(* PLC project Practical Work One, Rexroth ctrlX PLC Engineering ctrlX PLC 1.16.1, author Cedric Lenoir *)
(* stored: creationDateTime 2024-02-07T14:58:28.9317925, version 0.0, modificationDateTime 2024-02-07T14:56:44.3352338, organization HEVS *)
(* First Test for Practical Work One *)

TYPE UA_DigitalInput_32 : STRUCT
  Input_0_0 : BOOL;
  Input_0_1 : BOOL;
  Input_0_2 : BOOL;
  Input_0_3 : BOOL;
  Input_0_4 : BOOL;
  Input_0_5 : BOOL;
  Input_0_6 : BOOL;
  Input_0_7 : BOOL;
  Input_1_0 : BOOL;
  Input_1_1 : BOOL;
  Input_1_2 : BOOL;
  Input_1_3 : BOOL;
  Input_1_4 : BOOL;
  Input_1_5 : BOOL;
  Input_1_6 : BOOL;
  Input_1_7 : BOOL;
  Input_2_0 : BOOL;
  Input_2_1 : BOOL;
  Input_2_2 : BOOL;
  Input_2_3 : BOOL;
  Input_2_4 : BOOL;
  Input_2_5 : BOOL;
  Input_2_6 : BOOL;
  Input_2_7 : BOOL;
  Input_3_0 : BOOL;
  Input_3_1 : BOOL;
  Input_3_2 : BOOL;
  Input_3_3 : BOOL;
  Input_3_4 : BOOL;
  Input_3_5 : BOOL;
  Input_3_6 : BOOL;
  Input_3_7 : BOOL;
END_STRUCT;
END_TYPE

TYPE UA_DigitalOutput_32 : STRUCT
  Output_0_0 : BOOL;
  Output_0_1 : BOOL;
  Output_0_2 : BOOL;
  Output_0_3 : BOOL;
  Output_0_4 : BOOL;
  Output_0_5 : BOOL;
  Output_0_6 : BOOL;
  Output_0_7 : BOOL;
  Output_1_0 : BOOL;
  Output_1_1 : BOOL;
  Output_1_2 : BOOL;
  Output_1_3 : BOOL;
  Output_1_4 : BOOL;
  Output_1_5 : BOOL;
  Output_1_6 : BOOL;
  Output_1_7 : BOOL;
  Output_2_0 : BOOL;
  Output_2_1 : BOOL;
  Output_2_2 : BOOL;
  Output_2_3 : BOOL;
  Output_2_4 : BOOL;
  Output_2_5 : BOOL;
  Output_2_6 : BOOL;
  Output_2_7 : BOOL;
  Output_3_0 : BOOL;
  Output_3_1 : BOOL;
  Output_3_2 : BOOL;
  Output_3_3 : BOOL;
  Output_3_4 : BOOL;
  Output_3_5 : BOOL;
  Output_3_6 : BOOL;
  Output_3_7 : BOOL;
END_STRUCT;
END_TYPE

TYPE UA_ButtonAndSignal : STRUCT
  In_Estop : BOOL;
  In_Reset : BOOL;
  In_Start : BOOL;
  In_Stop : BOOL;
  Out_Idle : BOOL;
  Out_Execute : BOOL;
  Out_Stopped : BOOL;
END_STRUCT;
END_TYPE

TYPE UA_O300_DL : STRUCT
  Value : WORD;
  BCD1 : BOOL;
  Q : BOOL;
  A : BOOL;
END_STRUCT;
END_TYPE

TYPE UA_O300_ZL : STRUCT
  BCD1 : BOOL;
  Q : BOOL;
  A : BOOL;
END_STRUCT;
END_TYPE

TYPE UA_U300_D50 : STRUCT
  Value : DWORD;
  Scale : SINT;
  SSC1 : BOOL;
  SSC2 : BOOL;
  Q : BOOL;
  A : BOOL;
  SSC4 : BOOL;
END_STRUCT;
END_TYPE

(* www.hevs.ch Institut Systemes Industriels Project: Projet No: PW_01 Author: Cedric Lenoir Date: 2023 October 11 Summary: List of of components for a station of a conveyor. *)
TYPE ST_StationConveyor : STRUCT
  bButton : BOOL;
  bLed : BOOL;
  bSensor : BOOL;
END_STRUCT;
END_TYPE

(* www.hevs.ch Institut Systemes Industriels Project: Projet No: PW_01 Author: Cedric Lenoir Date: 2023 October 11 Summary: List of of components for a motor of a conveyor. *)
TYPE ST_BuzzerConveyor : STRUCT
  bActivate : BOOL;
  tTime : TIME := TIME#2s0ms;
END_STRUCT;
END_TYPE

(* www.hevs.ch Institut Systemes Industriels Project: Projet No: PW_01 Author: Cedric Lenoir Date: 2023 October 11 Summary: List of of components for a motor of a conveyor. *)
TYPE ST_MotorConveyor : STRUCT
  bK_ActivatePositiveDirection : BOOL;
  bK_ActivateNegativeDirection : BOOL;
END_STRUCT;
END_TYPE

TYPE ST_Conveyor : STRUCT
  StationOne : ST_StationConveyor;
  StationTwo : ST_StationConveyor;
  StationThree : ST_StationConveyor;
  StationOutput : ST_StationConveyor;
  Motor : ST_MotorConveyor;
  Buzzer : ST_BuzzerConveyor;
END_STRUCT;
END_TYPE

TYPE ST_HmiConveyor : STRUCT
  bStartConveyor : BOOL;
  bStopConveyor : BOOL;
END_STRUCT;
END_TYPE

TYPE UA_U300_P50 : STRUCT
  Value : DWORD;
  Scale : SINT;
  SSC1 : BOOL;
  SSC2 : BOOL;
  Q : BOOL;
  A : BOOL;
  SSC4 : BOOL;
END_STRUCT;
END_TYPE

TYPE UA_Schunk_mms : STRUCT
  Value : WORD;
END_STRUCT;
END_TYPE

TYPE UA_Balluf_bcm0002 : STRUCT
  Data_1 : REAL;
  Data_2 : REAL;
  Data_3 : REAL;
  Temperature : REAL;
  Status : DWORD;
END_STRUCT;
END_TYPE

TYPE UA_Festo : STRUCT
  SetOut : BOOL;
END_STRUCT;
END_TYPE

TYPE UA_AnalogIn : STRUCT
  IW_04 : WORD;
  IW_06 : WORD;
  IW_08 : WORD;
  IW_10 : WORD;
  IW_12 : WORD;
  IW_14 : WORD;
  IW_16 : WORD;
  IW_18 : WORD;
END_STRUCT;
END_TYPE

TYPE UA_AnalogOut : STRUCT
  QW_04 : WORD;
  QW_06 : WORD;
  QW_08 : WORD;
  QW_10 : WORD;
END_STRUCT;
END_TYPE

TYPE UA_AboxInterface : STRUCT
  uaButtonAndSignal : UA_ButtonAndSignal;
  uaAnalogIn : UA_AnalogIn;
  uaAnalogOut : UA_AnalogOut;
  uaDigitalIn : UA_DigitalInput_32;
  uaDigitalOut : UA_DigitalOutput_32;
  uaO300_DL_Optic : UA_O300_DL;
  uaO300_ZL_Optic : UA_O300_ZL;
  uaU300_D50_Sound : UA_U300_D50;
  uaU300_P50_Sound : UA_U300_P50;
  uaSchunk : UA_Schunk_mms;
  uaSchunkGripper : UA_Festo;
  uaAccelerometer : UA_Balluf_bcm0002;
END_STRUCT;
END_TYPE

TYPE ST_ConveyorTagsIn : STRUCT
  S1_Pb_Station_1 : BOOL;  (* %I0.0 *)
  S2_Pb_Station_2 : BOOL;  (* %I0.1 *)
  S3_Pb_Station_3 : BOOL;  (* %I0.2 *)
  S4_Pb_OutputConveyor : BOOL;  (* %I0.3 *)
  B1_SensorActive : BOOL;  (* %I0.4 *)
  B2_SensorActive : BOOL;  (* %I0.5 *)
  B3_SensorActive : BOOL;  (* %I0.6 *)
  B4_OutputConveyorFree : BOOL;  (* %I0.7 *)
END_STRUCT;
END_TYPE

TYPE ST_ConveyorTagsOut : STRUCT
  H1_LedStation_1 : BOOL;  (* %Q0.0 *)
  H2_LedStation_2 : BOOL;  (* %Q0.1 *)
  H3_LedStation_3 : BOOL;  (* %Q0.2 *)
  H4_LedOutputConveyor : BOOL;  (* %Q0.3 *)
  K1_DirectionOutput : BOOL;  (* %Q0.4 *)
  K2_DirectionH1 : BOOL;  (* %Q0.5 *)
  Buzzer : BOOL;  (* %Q0.6 *)
END_STRUCT;
END_TYPE

(* www.hevs.ch Institut Systemes Industriels Project: Projet No: PW_01 Author: Cedric Lenoir Date: 2023 October 11 Summary: PLC Hello World ! *)
PROGRAM PLC_PRG
  VAR
    iCount : INT := 3;
    TagIn : ST_ConveyorTagsIn;
    TagOut : ST_ConveyorTagsOut;
    rTrigStart : R_TRIG;
    rTrigStop : R_TRIG;
    tonBuzzer : TON;
  END_VAR

                    iCount := iCount + 1;

GetInput();

(*
	Declaration of all FB at the end of the code, this is a good practice.
	You can lose one cycle but the program is more readable.

    But !
    Triggers are exceptions:
        because the output .Q is only active in the current cycle
*)
rTrigStart(CLK:=GVL_Abox.uaAboxInterface.uaButtonAndSignal.In_Start);
rTrigStop(CLK:=GVL_Abox.uaAboxInterface.uaButtonAndSignal.In_Stop);

IF rTrigStart.Q THEN
	TagOut.K1_DirectionOutput := TRUE;
END_IF

IF rTrigStop.Q THEN
	TagOut.K1_DirectionOutput := FALSE;
END_IF

// If Start activated for more than 3 seconds, then Buzzer
tonBuzzer(IN := GVL_Abox.uaAboxInterface.uaButtonAndSignal.In_Start,
	      PT := T#3S);
		  
TagOut.Buzzer := tonBuzzer.Q;

SetOutput();
                  

METHOD GetInput
                          TagIn.S1_Pb_Station_1 := GVL_Abox.uaAboxInterface.uaDigitalIn.Input_0_0;
TagIn.S2_Pb_Station_2 := GVL_Abox.uaAboxInterface.uaDigitalIn.Input_0_1;
TagIn.S3_Pb_Station_3 := GVL_Abox.uaAboxInterface.uaDigitalIn.Input_0_2;
TagIn.S4_Pb_OutputConveyor := GVL_Abox.uaAboxInterface.uaDigitalIn.Input_0_3;

TagIn.B1_SensorActive := GVL_Abox.uaAboxInterface.uaDigitalIn.Input_0_4;
TagIn.B2_SensorActive := GVL_Abox.uaAboxInterface.uaDigitalIn.Input_0_5;
TagIn.B3_SensorActive := GVL_Abox.uaAboxInterface.uaDigitalIn.Input_0_6;
TagIn.B4_OutputConveyorFree := GVL_Abox.uaAboxInterface.uaDigitalIn.Input_0_7;
                        
END_METHOD

METHOD SetOutput
                          GVL_Abox.uaAboxInterface.uaDigitalOut.Output_0_0 := TagOut.H1_LedStation_1;
GVL_Abox.uaAboxInterface.uaDigitalOut.Output_0_1 := TagOut.H2_LedStation_2;
GVL_Abox.uaAboxInterface.uaDigitalOut.Output_0_2 := TagOut.H3_LedStation_3;
GVL_Abox.uaAboxInterface.uaDigitalOut.Output_0_3 := TagOut.H4_LedOutputConveyor;
GVL_Abox.uaAboxInterface.uaDigitalOut.Output_0_4 := TagOut.K1_DirectionOutput;
GVL_Abox.uaAboxInterface.uaDigitalOut.Output_0_5 := TagOut.K2_DirectionH1;
GVL_Abox.uaAboxInterface.uaDigitalOut.Output_0_6 := TagOut.Buzzer;
                        
END_METHOD
END_PROGRAM

PROGRAM PRG_MapBox
  VAR
    UA_ReadCounterFromStation : DINT;  (* Write from Siemens to ctrX Core Used to check if read is running *)
    UA_ButtonAndSignal_In_Estop : BOOL;
    UA_ButtonAndSignal_In_Reset : BOOL;
    UA_ButtonAndSignal_In_Start : BOOL;
    UA_ButtonAndSignal_In_Stop : BOOL;
    UA_Balluf_bcm0002_Data_1 : REAL;
    UA_Balluf_bcm0002_Data_2 : REAL;
    UA_Balluf_bcm0002_Data_3 : REAL;
    UA_Balluf_bcm0002_Temperature : REAL;
    UA_Balluf_bcm0002_Status : DWORD;
    UA_Festo_SetOut : BOOL;
    UA_O300_DL_Value : WORD;
    UA_O300_DL_BCD1 : BOOL;
    UA_O300_DL_Q : BOOL;
    UA_O300_DL_A : BOOL;
    UA_O300_ZL_BCD1 : BOOL;
    UA_O300_ZL_Q : BOOL;
    UA_O300_ZL_A : BOOL;
    UA_U300_D50_Value : DWORD;
    UA_U300_D50_Scale : SINT;
    UA_U300_D50_SSC1 : BOOL;
    UA_U300_D50_SSC2 : BOOL;
    UA_U300_D50_Q : BOOL;
    UA_U300_D50_A : BOOL;
    UA_U300_D50_SSC4 : BOOL;
    UA_U300_P50_Value : DWORD;
    UA_U300_P50_Scale : SINT;
    UA_U300_P50_SSC1 : BOOL;
    UA_U300_P50_SSC2 : BOOL;
    UA_U300_P50_Q : BOOL;
    UA_U300_P50_A : BOOL;
    UA_U300_P50_SSC4 : BOOL;
    UA_DigitalInput_32_Input_0_0 : BOOL;
    UA_DigitalInput_32_Input_0_1 : BOOL;
    UA_DigitalInput_32_Input_0_2 : BOOL;
    UA_DigitalInput_32_Input_0_3 : BOOL;
    UA_DigitalInput_32_Input_0_4 : BOOL;
    UA_DigitalInput_32_Input_0_5 : BOOL;
    UA_DigitalInput_32_Input_0_6 : BOOL;
    UA_DigitalInput_32_Input_0_7 : BOOL;
    UA_DigitalInput_32_Input_1_0 : BOOL;
    UA_DigitalInput_32_Input_1_1 : BOOL;
    UA_DigitalInput_32_Input_1_2 : BOOL;
    UA_DigitalInput_32_Input_1_3 : BOOL;
    UA_DigitalInput_32_Input_1_4 : BOOL;
    UA_DigitalInput_32_Input_1_5 : BOOL;
    UA_DigitalInput_32_Input_1_6 : BOOL;
    UA_DigitalInput_32_Input_1_7 : BOOL;
    UA_DigitalInput_32_Input_2_0 : BOOL;
    UA_DigitalInput_32_Input_2_1 : BOOL;
    UA_DigitalInput_32_Input_2_2 : BOOL;
    UA_DigitalInput_32_Input_2_3 : BOOL;
    UA_DigitalInput_32_Input_2_4 : BOOL;
    UA_DigitalInput_32_Input_2_5 : BOOL;
    UA_DigitalInput_32_Input_2_6 : BOOL;
    UA_DigitalInput_32_Input_2_7 : BOOL;
    UA_DigitalInput_32_Input_3_0 : BOOL;
    UA_DigitalInput_32_Input_3_1 : BOOL;
    UA_DigitalInput_32_Input_3_2 : BOOL;
    UA_DigitalInput_32_Input_3_3 : BOOL;
    UA_DigitalInput_32_Input_3_4 : BOOL;
    UA_DigitalInput_32_Input_3_5 : BOOL;
    UA_DigitalInput_32_Input_3_6 : BOOL;
    UA_DigitalInput_32_Input_3_7 : BOOL;
    UA_WriteCounterToStation : DINT;  (* Siemens Read from ctrX Core Used to check if write is running *)
    UA_ButtonAndSignal_Out_Idle : BOOL;
    UA_ButtonAndSignal_Out_Execute : BOOL;
    UA_ButtonAndSignal_Out_Stopped : BOOL;
    UA_Schunk_mms_Value : WORD;
    UA_DigitalOutput_32_Output_0_0 : BOOL;
    UA_DigitalOutput_32_Output_0_1 : BOOL;
    UA_DigitalOutput_32_Output_0_2 : BOOL;
    UA_DigitalOutput_32_Output_0_3 : BOOL;
    UA_DigitalOutput_32_Output_0_4 : BOOL;
    UA_DigitalOutput_32_Output_0_5 : BOOL;
    UA_DigitalOutput_32_Output_0_6 : BOOL;
    UA_DigitalOutput_32_Output_0_7 : BOOL;
    UA_DigitalOutput_32_Output_1_0 : BOOL;
    UA_DigitalOutput_32_Output_1_1 : BOOL;
    UA_DigitalOutput_32_Output_1_2 : BOOL;
    UA_DigitalOutput_32_Output_1_3 : BOOL;
    UA_DigitalOutput_32_Output_1_4 : BOOL;
    UA_DigitalOutput_32_Output_1_5 : BOOL;
    UA_DigitalOutput_32_Output_1_6 : BOOL;
    UA_DigitalOutput_32_Output_1_7 : BOOL;
    UA_DigitalOutput_32_Output_2_0 : BOOL;
    UA_DigitalOutput_32_Output_2_1 : BOOL;
    UA_DigitalOutput_32_Output_2_2 : BOOL;
    UA_DigitalOutput_32_Output_2_3 : BOOL;
    UA_DigitalOutput_32_Output_2_4 : BOOL;
    UA_DigitalOutput_32_Output_2_5 : BOOL;
    UA_DigitalOutput_32_Output_2_6 : BOOL;
    UA_DigitalOutput_32_Output_2_7 : BOOL;
    UA_DigitalOutput_32_Output_3_0 : BOOL;
    UA_DigitalOutput_32_Output_3_1 : BOOL;
    UA_DigitalOutput_32_Output_3_2 : BOOL;
    UA_DigitalOutput_32_Output_3_3 : BOOL;
    UA_DigitalOutput_32_Output_3_4 : BOOL;
    UA_DigitalOutput_32_Output_3_5 : BOOL;
    UA_DigitalOutput_32_Output_3_6 : BOOL;
    UA_DigitalOutput_32_Output_3_7 : BOOL;
  END_VAR

                        (*
        Values from Profinet Station
    *)
    
    // Get Value from Profinet Station with UA Client Write
	GVL_Abox.uaAboxInterface.uaButtonAndSignal.In_Estop     := UA_ButtonAndSignal_In_Estop;
	GVL_Abox.uaAboxInterface.uaButtonAndSignal.In_Reset     := UA_ButtonAndSignal_In_Reset;
	GVL_Abox.uaAboxInterface.uaButtonAndSignal.In_Start     := UA_ButtonAndSignal_In_Start;
	GVL_Abox.uaAboxInterface.uaButtonAndSignal.In_Stop      := UA_ButtonAndSignal_In_Stop;
    // Values from Balluff accelerometer
    GVL_Abox.uaAboxInterface.uaAccelerometer.Data_1         := UA_Balluf_bcm0002_Data_1;
    GVL_Abox.uaAboxInterface.uaAccelerometer.Data_2         := UA_Balluf_bcm0002_Data_1;
    GVL_Abox.uaAboxInterface.uaAccelerometer.Data_3         := UA_Balluf_bcm0002_Data_1;
    GVL_Abox.uaAboxInterface.uaAccelerometer.Status         := UA_Balluf_bcm0002_Status;
    GVL_Abox.uaAboxInterface.uaAccelerometer.Temperature    := UA_Balluf_bcm0002_Temperature;

    // Values from Baumer O300 DL
    GVL_Abox.uaAboxInterface.uaO300_DL_Optic.Value          := UA_O300_DL_Value;                
    GVL_Abox.uaAboxInterface.uaO300_DL_Optic.A              := UA_O300_DL_A;                
    GVL_Abox.uaAboxInterface.uaO300_DL_Optic.Q              := UA_O300_DL_Q;                
    GVL_Abox.uaAboxInterface.uaO300_DL_Optic.BCD1           := UA_O300_DL_BCD1;                

    // Values from Baumer O300 ZL                
    GVL_Abox.uaAboxInterface.uaO300_ZL_Optic.A              := UA_O300_ZL_A;                
    GVL_Abox.uaAboxInterface.uaO300_ZL_Optic.Q              := UA_O300_ZL_Q;                
    GVL_Abox.uaAboxInterface.uaO300_ZL_Optic.BCD1           := UA_O300_ZL_BCD1;                

    // Values from Baumer U300 D50
    GVL_Abox.uaAboxInterface.uaU300_D50_Sound.Value         := UA_U300_D50_Value;  
    GVL_Abox.uaAboxInterface.uaU300_D50_Sound.A             := UA_U300_D50_A;  
    GVL_Abox.uaAboxInterface.uaU300_D50_Sound.Q             := UA_U300_D50_Q;  
    GVL_Abox.uaAboxInterface.uaU300_D50_Sound.Scale         := UA_U300_D50_Scale;  
    GVL_Abox.uaAboxInterface.uaU300_D50_Sound.SSC1          := UA_U300_D50_SSC1;  
    GVL_Abox.uaAboxInterface.uaU300_D50_Sound.SSC2          := UA_U300_D50_SSC2;  
    GVL_Abox.uaAboxInterface.uaU300_D50_Sound.SSC4          := UA_U300_D50_SSC4;  
    
    // Values from Baumer U300 P50
    GVL_Abox.uaAboxInterface.uaU300_P50_Sound.Value         := UA_U300_P50_Value;  
    GVL_Abox.uaAboxInterface.uaU300_P50_Sound.A             := UA_U300_P50_A;  
    GVL_Abox.uaAboxInterface.uaU300_P50_Sound.Q             := UA_U300_P50_Q;  
    GVL_Abox.uaAboxInterface.uaU300_P50_Sound.Scale         := UA_U300_P50_Scale;  
    GVL_Abox.uaAboxInterface.uaU300_P50_Sound.SSC1          := UA_U300_P50_SSC1;  
    GVL_Abox.uaAboxInterface.uaU300_P50_Sound.SSC2          := UA_U300_P50_SSC2;  
    GVL_Abox.uaAboxInterface.uaU300_P50_Sound.SSC4          := UA_U300_P50_SSC4;  
    
    // Values from Gripper sensor
    GVL_Abox.uaAboxInterface.uaSchunk.Value                 := UA_Schunk_mms_Value;  
    
    // Get 32 Digital Input
    GVL_Abox.uaAboxInterface.uaDigitalIn.Input_0_0          := UA_DigitalInput_32_Input_0_0;
    GVL_Abox.uaAboxInterface.uaDigitalIn.Input_0_1          := UA_DigitalInput_32_Input_0_1;
    GVL_Abox.uaAboxInterface.uaDigitalIn.Input_0_2          := UA_DigitalInput_32_Input_0_2;
    GVL_Abox.uaAboxInterface.uaDigitalIn.Input_0_3          := UA_DigitalInput_32_Input_0_3;
    GVL_Abox.uaAboxInterface.uaDigitalIn.Input_0_4          := UA_DigitalInput_32_Input_0_4;
    GVL_Abox.uaAboxInterface.uaDigitalIn.Input_0_5          := UA_DigitalInput_32_Input_0_5;
    GVL_Abox.uaAboxInterface.uaDigitalIn.Input_0_6          := UA_DigitalInput_32_Input_0_6;
    GVL_Abox.uaAboxInterface.uaDigitalIn.Input_0_7          := UA_DigitalInput_32_Input_0_7;
    GVL_Abox.uaAboxInterface.uaDigitalIn.Input_1_0          := UA_DigitalInput_32_Input_1_0;
    GVL_Abox.uaAboxInterface.uaDigitalIn.Input_1_1          := UA_DigitalInput_32_Input_1_1;
    GVL_Abox.uaAboxInterface.uaDigitalIn.Input_1_2          := UA_DigitalInput_32_Input_1_2;
    GVL_Abox.uaAboxInterface.uaDigitalIn.Input_1_3          := UA_DigitalInput_32_Input_1_3;
    GVL_Abox.uaAboxInterface.uaDigitalIn.Input_1_4          := UA_DigitalInput_32_Input_1_4;
    GVL_Abox.uaAboxInterface.uaDigitalIn.Input_1_5          := UA_DigitalInput_32_Input_1_5;
    GVL_Abox.uaAboxInterface.uaDigitalIn.Input_1_6          := UA_DigitalInput_32_Input_1_6;
    GVL_Abox.uaAboxInterface.uaDigitalIn.Input_1_7          := UA_DigitalInput_32_Input_1_7;
    GVL_Abox.uaAboxInterface.uaDigitalIn.Input_2_0          := UA_DigitalInput_32_Input_2_0;
    GVL_Abox.uaAboxInterface.uaDigitalIn.Input_2_1          := UA_DigitalInput_32_Input_2_1;
    GVL_Abox.uaAboxInterface.uaDigitalIn.Input_2_2          := UA_DigitalInput_32_Input_2_2;
    GVL_Abox.uaAboxInterface.uaDigitalIn.Input_2_3          := UA_DigitalInput_32_Input_2_3;
    GVL_Abox.uaAboxInterface.uaDigitalIn.Input_2_4          := UA_DigitalInput_32_Input_2_4;
    GVL_Abox.uaAboxInterface.uaDigitalIn.Input_2_5          := UA_DigitalInput_32_Input_2_5;
    GVL_Abox.uaAboxInterface.uaDigitalIn.Input_2_6          := UA_DigitalInput_32_Input_2_6;
    GVL_Abox.uaAboxInterface.uaDigitalIn.Input_2_7          := UA_DigitalInput_32_Input_2_7;
    GVL_Abox.uaAboxInterface.uaDigitalIn.Input_3_0          := UA_DigitalInput_32_Input_3_0;
    GVL_Abox.uaAboxInterface.uaDigitalIn.Input_3_1          := UA_DigitalInput_32_Input_3_1;
    GVL_Abox.uaAboxInterface.uaDigitalIn.Input_3_2          := UA_DigitalInput_32_Input_3_2;
    GVL_Abox.uaAboxInterface.uaDigitalIn.Input_3_3          := UA_DigitalInput_32_Input_3_3;
    GVL_Abox.uaAboxInterface.uaDigitalIn.Input_3_4          := UA_DigitalInput_32_Input_3_4;
    GVL_Abox.uaAboxInterface.uaDigitalIn.Input_3_5          := UA_DigitalInput_32_Input_3_5;
    GVL_Abox.uaAboxInterface.uaDigitalIn.Input_3_6          := UA_DigitalInput_32_Input_3_6;
    GVL_Abox.uaAboxInterface.uaDigitalIn.Input_3_7          := UA_DigitalInput_32_Input_3_7;
    
    (*
        Values to Profinet Station
    *)
	UA_WriteCounterToStation := UA_WriteCounterToStation + 1;

    // Set Visual Signals
	UA_ButtonAndSignal_Out_Execute 	:= GVL_Abox.uaAboxInterface.uaButtonAndSignal.Out_Execute;
	UA_ButtonAndSignal_Out_Idle 	:= GVL_Abox.uaAboxInterface.uaButtonAndSignal.Out_Idle;
	UA_ButtonAndSignal_Out_Stopped	:= GVL_Abox.uaAboxInterface.uaButtonAndSignal.Out_Stopped;
    
    // Set Gripper value
    UA_Festo_SetOut                 := GVL_Abox.uaAboxInterface.uaSchunkGripper.SetOut;
    
    // Set 32 digital outputs
    UA_DigitalOutput_32_Output_0_0  := GVL_Abox.uaAboxInterface.uaDigitalOut.Output_0_0;
    UA_DigitalOutput_32_Output_0_1  := GVL_Abox.uaAboxInterface.uaDigitalOut.Output_0_1;
    UA_DigitalOutput_32_Output_0_2  := GVL_Abox.uaAboxInterface.uaDigitalOut.Output_0_2;
    UA_DigitalOutput_32_Output_0_3  := GVL_Abox.uaAboxInterface.uaDigitalOut.Output_0_3;
    UA_DigitalOutput_32_Output_0_4  := GVL_Abox.uaAboxInterface.uaDigitalOut.Output_0_4;
    UA_DigitalOutput_32_Output_0_5  := GVL_Abox.uaAboxInterface.uaDigitalOut.Output_0_5;
    UA_DigitalOutput_32_Output_0_6  := GVL_Abox.uaAboxInterface.uaDigitalOut.Output_0_6;
    UA_DigitalOutput_32_Output_0_7  := GVL_Abox.uaAboxInterface.uaDigitalOut.Output_0_7;
    UA_DigitalOutput_32_Output_1_0  := GVL_Abox.uaAboxInterface.uaDigitalOut.Output_1_0;
    UA_DigitalOutput_32_Output_1_1  := GVL_Abox.uaAboxInterface.uaDigitalOut.Output_1_1;
    UA_DigitalOutput_32_Output_1_2  := GVL_Abox.uaAboxInterface.uaDigitalOut.Output_1_2;
    UA_DigitalOutput_32_Output_1_3  := GVL_Abox.uaAboxInterface.uaDigitalOut.Output_1_3;
    UA_DigitalOutput_32_Output_1_4  := GVL_Abox.uaAboxInterface.uaDigitalOut.Output_1_4;
    UA_DigitalOutput_32_Output_1_5  := GVL_Abox.uaAboxInterface.uaDigitalOut.Output_1_5;
    UA_DigitalOutput_32_Output_1_6  := GVL_Abox.uaAboxInterface.uaDigitalOut.Output_1_6;
    UA_DigitalOutput_32_Output_1_7  := GVL_Abox.uaAboxInterface.uaDigitalOut.Output_1_7;
    UA_DigitalOutput_32_Output_2_0  := GVL_Abox.uaAboxInterface.uaDigitalOut.Output_2_0;
    UA_DigitalOutput_32_Output_2_1  := GVL_Abox.uaAboxInterface.uaDigitalOut.Output_2_1;
    UA_DigitalOutput_32_Output_2_2  := GVL_Abox.uaAboxInterface.uaDigitalOut.Output_2_2;
    UA_DigitalOutput_32_Output_2_3  := GVL_Abox.uaAboxInterface.uaDigitalOut.Output_2_3;
    UA_DigitalOutput_32_Output_2_4  := GVL_Abox.uaAboxInterface.uaDigitalOut.Output_2_4;
    UA_DigitalOutput_32_Output_2_5  := GVL_Abox.uaAboxInterface.uaDigitalOut.Output_2_5;
    UA_DigitalOutput_32_Output_2_6  := GVL_Abox.uaAboxInterface.uaDigitalOut.Output_2_6;
    UA_DigitalOutput_32_Output_2_7  := GVL_Abox.uaAboxInterface.uaDigitalOut.Output_2_7;
    UA_DigitalOutput_32_Output_3_0  := GVL_Abox.uaAboxInterface.uaDigitalOut.Output_3_0;
    UA_DigitalOutput_32_Output_3_1  := GVL_Abox.uaAboxInterface.uaDigitalOut.Output_3_1;
    UA_DigitalOutput_32_Output_3_2  := GVL_Abox.uaAboxInterface.uaDigitalOut.Output_3_2;
    UA_DigitalOutput_32_Output_3_3  := GVL_Abox.uaAboxInterface.uaDigitalOut.Output_3_3;
    UA_DigitalOutput_32_Output_3_4  := GVL_Abox.uaAboxInterface.uaDigitalOut.Output_3_4;
    UA_DigitalOutput_32_Output_3_5  := GVL_Abox.uaAboxInterface.uaDigitalOut.Output_3_5;
    UA_DigitalOutput_32_Output_3_6  := GVL_Abox.uaAboxInterface.uaDigitalOut.Output_3_6;
    UA_DigitalOutput_32_Output_3_7  := GVL_Abox.uaAboxInterface.uaDigitalOut.Output_3_7;
    
PRG_CHECK_IO();
                  
END_PROGRAM

PROGRAM PRG_CHECK_IO
  VAR
    testButton_1 : BOOL;
    testButton_2 : BOOL;
    testButton_3 : BOOL;
    clignote : TON;
    changeMeSlow : BOOL;
    clignoteSlow : TON;
    changeMe : BOOL;
    NotResetTest : BOOL := TRUE;
  END_VAR

                    testButton_1 := GVL_Abox.uaAboxInterface.uaButtonAndSignal.In_Reset;
testButton_2 := GVL_Abox.uaAboxInterface.uaButtonAndSignal.In_Start;
testButton_3 := GVL_Abox.uaAboxInterface.uaButtonAndSignal.In_Stop;

IF GVL_Abox.uaAboxInterface.uaButtonAndSignal.In_Reset AND
   NotResetTest										   THEN
	NotResetTest := FALSE;
	
    GVL_Abox.uaAboxInterface.uaSchunkGripper.SetOut := FALSE;
    
    GVL_Abox.uaAboxInterface.uaButtonAndSignal.Out_Execute := FALSE;	
    GVL_Abox.uaAboxInterface.uaButtonAndSignal.Out_Idle := FALSE;	
    GVL_Abox.uaAboxInterface.uaButtonAndSignal.Out_Stopped := FALSE;	

    GVL_Abox.uaAboxInterface.uaDigitalOut.Output_0_0 := FALSE;
    GVL_Abox.uaAboxInterface.uaDigitalOut.Output_0_1 := FALSE;
    GVL_Abox.uaAboxInterface.uaDigitalOut.Output_0_2 := FALSE;
    GVL_Abox.uaAboxInterface.uaDigitalOut.Output_0_3 := FALSE;
    GVL_Abox.uaAboxInterface.uaDigitalOut.Output_0_4 := FALSE;
    GVL_Abox.uaAboxInterface.uaDigitalOut.Output_0_5 := FALSE;
    GVL_Abox.uaAboxInterface.uaDigitalOut.Output_0_6 := FALSE;
    GVL_Abox.uaAboxInterface.uaDigitalOut.Output_0_7 := FALSE;
    
    GVL_Abox.uaAboxInterface.uaDigitalOut.Output_1_0 := FALSE;
    GVL_Abox.uaAboxInterface.uaDigitalOut.Output_1_1 := FALSE;
    GVL_Abox.uaAboxInterface.uaDigitalOut.Output_1_2 := FALSE;
    GVL_Abox.uaAboxInterface.uaDigitalOut.Output_1_3 := FALSE;
    GVL_Abox.uaAboxInterface.uaDigitalOut.Output_1_4 := FALSE;
    GVL_Abox.uaAboxInterface.uaDigitalOut.Output_1_5 := FALSE;
    GVL_Abox.uaAboxInterface.uaDigitalOut.Output_1_6 := FALSE;
    GVL_Abox.uaAboxInterface.uaDigitalOut.Output_1_7 := FALSE;
    
    GVL_Abox.uaAboxInterface.uaDigitalOut.Output_2_0 := FALSE;
    GVL_Abox.uaAboxInterface.uaDigitalOut.Output_2_1 := FALSE;
    GVL_Abox.uaAboxInterface.uaDigitalOut.Output_2_2 := FALSE;
    GVL_Abox.uaAboxInterface.uaDigitalOut.Output_2_3 := FALSE;
    GVL_Abox.uaAboxInterface.uaDigitalOut.Output_2_4 := FALSE;
    GVL_Abox.uaAboxInterface.uaDigitalOut.Output_2_5 := FALSE;
    GVL_Abox.uaAboxInterface.uaDigitalOut.Output_2_6 := FALSE;
    GVL_Abox.uaAboxInterface.uaDigitalOut.Output_2_7 := FALSE;

    GVL_Abox.uaAboxInterface.uaDigitalOut.Output_3_0 := FALSE;
    GVL_Abox.uaAboxInterface.uaDigitalOut.Output_3_1 := FALSE;
    GVL_Abox.uaAboxInterface.uaDigitalOut.Output_3_2 := FALSE;
    GVL_Abox.uaAboxInterface.uaDigitalOut.Output_3_3 := FALSE;
    GVL_Abox.uaAboxInterface.uaDigitalOut.Output_3_4 := FALSE;
    GVL_Abox.uaAboxInterface.uaDigitalOut.Output_3_5 := FALSE;
    GVL_Abox.uaAboxInterface.uaDigitalOut.Output_3_6 := FALSE;
    GVL_Abox.uaAboxInterface.uaDigitalOut.Output_3_7 := FALSE;	
END_IF

IF GVL_Abox.uaAboxInterface.uaButtonAndSignal.In_Reset AND
   GVL_Abox.uaAboxInterface.uaButtonAndSignal.In_Start AND
   GVL_Abox.uaAboxInterface.uaButtonAndSignal.In_Stop  THEN
	NotResetTest := TRUE;
END_IF


IF NotResetTest THEN 
	
	// Quick Blink
	clignote(IN := changeMe,
			 PT := T#500MS);
			 
	IF clignote.Q THEN
		changeMe := FALSE;
	ELSE
		changeMe := TRUE;
	END_IF

	// Slow Blink
	clignoteSlow(IN := changeMeSlow,
			 	 PT := T#2500MS);
			 
	IF clignoteSlow.Q THEN
		changeMeSlow := FALSE;
	ELSE
		changeMeSlow := TRUE;
	END_IF
	
	IF (NOT GVL_Abox.uaAboxInterface.uaSchunkGripper.SetOut) AND clignoteSlow.Q THEN
		GVL_Abox.uaAboxInterface.uaSchunkGripper.SetOut := TRUE;
	ELSIF GVL_Abox.uaAboxInterface.uaSchunkGripper.SetOut AND clignoteSlow.Q THEN
		GVL_Abox.uaAboxInterface.uaSchunkGripper.SetOut := FALSE;
	END_IF
	
	IF (NOT GVL_Abox.uaAboxInterface.uaDigitalOut.Output_0_0) AND clignote.Q THEN
		GVL_Abox.uaAboxInterface.uaButtonAndSignal.Out_Execute := TRUE;	
		GVL_Abox.uaAboxInterface.uaButtonAndSignal.Out_Idle := TRUE;	
		GVL_Abox.uaAboxInterface.uaButtonAndSignal.Out_Stopped := TRUE;	
	
		GVL_Abox.uaAboxInterface.uaDigitalOut.Output_0_0 := TRUE;
		GVL_Abox.uaAboxInterface.uaDigitalOut.Output_0_1 := TRUE;
		GVL_Abox.uaAboxInterface.uaDigitalOut.Output_0_2 := TRUE;
		GVL_Abox.uaAboxInterface.uaDigitalOut.Output_0_3 := TRUE;
		GVL_Abox.uaAboxInterface.uaDigitalOut.Output_0_4 := TRUE;
		GVL_Abox.uaAboxInterface.uaDigitalOut.Output_0_5 := TRUE;
		GVL_Abox.uaAboxInterface.uaDigitalOut.Output_0_6 := TRUE;
		GVL_Abox.uaAboxInterface.uaDigitalOut.Output_0_7 := TRUE;
		
		GVL_Abox.uaAboxInterface.uaDigitalOut.Output_1_0 := TRUE;
		GVL_Abox.uaAboxInterface.uaDigitalOut.Output_1_1 := TRUE;
		GVL_Abox.uaAboxInterface.uaDigitalOut.Output_1_2 := TRUE;
		GVL_Abox.uaAboxInterface.uaDigitalOut.Output_1_3 := TRUE;
		GVL_Abox.uaAboxInterface.uaDigitalOut.Output_1_4 := TRUE;
		GVL_Abox.uaAboxInterface.uaDigitalOut.Output_1_5 := TRUE;
		GVL_Abox.uaAboxInterface.uaDigitalOut.Output_1_6 := TRUE;
		GVL_Abox.uaAboxInterface.uaDigitalOut.Output_1_7 := TRUE;
		
		GVL_Abox.uaAboxInterface.uaDigitalOut.Output_2_0 := TRUE;
		GVL_Abox.uaAboxInterface.uaDigitalOut.Output_2_1 := TRUE;
		GVL_Abox.uaAboxInterface.uaDigitalOut.Output_2_2 := TRUE;
		GVL_Abox.uaAboxInterface.uaDigitalOut.Output_2_3 := TRUE;
		GVL_Abox.uaAboxInterface.uaDigitalOut.Output_2_4 := TRUE;
		GVL_Abox.uaAboxInterface.uaDigitalOut.Output_2_5 := TRUE;
		GVL_Abox.uaAboxInterface.uaDigitalOut.Output_2_6 := TRUE;
		GVL_Abox.uaAboxInterface.uaDigitalOut.Output_2_7 := TRUE;

		GVL_Abox.uaAboxInterface.uaDigitalOut.Output_3_0 := TRUE;
		GVL_Abox.uaAboxInterface.uaDigitalOut.Output_3_1 := TRUE;
		GVL_Abox.uaAboxInterface.uaDigitalOut.Output_3_2 := TRUE;
		GVL_Abox.uaAboxInterface.uaDigitalOut.Output_3_3 := TRUE;
		GVL_Abox.uaAboxInterface.uaDigitalOut.Output_3_4 := TRUE;
		GVL_Abox.uaAboxInterface.uaDigitalOut.Output_3_5 := TRUE;
		GVL_Abox.uaAboxInterface.uaDigitalOut.Output_3_6 := TRUE;
		GVL_Abox.uaAboxInterface.uaDigitalOut.Output_3_7 := TRUE;
	ELSIF GVL_Abox.uaAboxInterface.uaDigitalOut.Output_0_0 AND clignote.Q THEN
		GVL_Abox.uaAboxInterface.uaButtonAndSignal.Out_Execute := FALSE;	
		GVL_Abox.uaAboxInterface.uaButtonAndSignal.Out_Idle := FALSE;	
		GVL_Abox.uaAboxInterface.uaButtonAndSignal.Out_Stopped := FALSE;	

		GVL_Abox.uaAboxInterface.uaDigitalOut.Output_0_0 := FALSE;
		GVL_Abox.uaAboxInterface.uaDigitalOut.Output_0_1 := FALSE;
		GVL_Abox.uaAboxInterface.uaDigitalOut.Output_0_2 := FALSE;
		GVL_Abox.uaAboxInterface.uaDigitalOut.Output_0_3 := FALSE;
		GVL_Abox.uaAboxInterface.uaDigitalOut.Output_0_4 := FALSE;
		GVL_Abox.uaAboxInterface.uaDigitalOut.Output_0_5 := FALSE;
		GVL_Abox.uaAboxInterface.uaDigitalOut.Output_0_6 := FALSE;
		GVL_Abox.uaAboxInterface.uaDigitalOut.Output_0_7 := FALSE;
		
		GVL_Abox.uaAboxInterface.uaDigitalOut.Output_1_0 := FALSE;
		GVL_Abox.uaAboxInterface.uaDigitalOut.Output_1_1 := FALSE;
		GVL_Abox.uaAboxInterface.uaDigitalOut.Output_1_2 := FALSE;
		GVL_Abox.uaAboxInterface.uaDigitalOut.Output_1_3 := FALSE;
		GVL_Abox.uaAboxInterface.uaDigitalOut.Output_1_4 := FALSE;
		GVL_Abox.uaAboxInterface.uaDigitalOut.Output_1_5 := FALSE;
		GVL_Abox.uaAboxInterface.uaDigitalOut.Output_1_6 := FALSE;
		GVL_Abox.uaAboxInterface.uaDigitalOut.Output_1_7 := FALSE;
		
		GVL_Abox.uaAboxInterface.uaDigitalOut.Output_2_0 := FALSE;
		GVL_Abox.uaAboxInterface.uaDigitalOut.Output_2_1 := FALSE;
		GVL_Abox.uaAboxInterface.uaDigitalOut.Output_2_2 := FALSE;
		GVL_Abox.uaAboxInterface.uaDigitalOut.Output_2_3 := FALSE;
		GVL_Abox.uaAboxInterface.uaDigitalOut.Output_2_4 := FALSE;
		GVL_Abox.uaAboxInterface.uaDigitalOut.Output_2_5 := FALSE;
		GVL_Abox.uaAboxInterface.uaDigitalOut.Output_2_6 := FALSE;
		GVL_Abox.uaAboxInterface.uaDigitalOut.Output_2_7 := FALSE;

		GVL_Abox.uaAboxInterface.uaDigitalOut.Output_3_0 := FALSE;
		GVL_Abox.uaAboxInterface.uaDigitalOut.Output_3_1 := FALSE;
		GVL_Abox.uaAboxInterface.uaDigitalOut.Output_3_2 := FALSE;
		GVL_Abox.uaAboxInterface.uaDigitalOut.Output_3_3 := FALSE;
		GVL_Abox.uaAboxInterface.uaDigitalOut.Output_3_4 := FALSE;
		GVL_Abox.uaAboxInterface.uaDigitalOut.Output_3_5 := FALSE;
		GVL_Abox.uaAboxInterface.uaDigitalOut.Output_3_6 := FALSE;
		GVL_Abox.uaAboxInterface.uaDigitalOut.Output_3_7 := FALSE;
	END_IF;
END_IF
                  
END_PROGRAM

CONFIGURATION PracticalWork_01
  RESOURCE BaseInterfaceUa ON PLC
    {attribute 'qualified_only'}
    VAR_GLOBAL  (* GVL_Abox *)
      uaAboxInterface : UA_AboxInterface;
    END_VAR
    {attribute 'qualified_only'}
    VAR_GLOBAL  (* GVL_Unit *)
      myConveyor : ST_Conveyor;
      myHmi : ST_HmiConveyor;
    END_VAR
    TASK MainTask(INTERVAL := T#10ms, PRIORITY := 30);
    PROGRAM PLC_PRG WITH MainTask : PLC_PRG;
    PROGRAM PRG_MapBox WITH MainTask : PRG_MapBox;
  END_RESOURCE
END_CONFIGURATION

CONFIGURATION Realtime_Data
END_CONFIGURATION
